TEXTLIST TextList
  0 = 'Sistem' | Türkçe: 'Sistem' | İngilizce: 'System'
  1 = 'Dil Seçeneği' | Türkçe: 'Dil Seçeneği' | İngilizce: 'Languages'
  2 = 'Ana Sayfa' | Türkçe: 'Ana Sayfa' | İngilizce: 'Home Page'
  3 = 'İngilizce' | Türkçe: 'İngilizce' | İngilizce: 'English'
  4 = 'Türkçe' | Türkçe: 'Türkçe' | İngilizce: 'Turkish'
   = ''
END_TEXTLIST

(* stored: Version 1.1.0.1, ProductVersion 3.1.4024.4
   TextList TextList: Id {07723166-985a-47af-92d4-fcd1ae42f531} *)
